{attribute addProperty BoxType "EL2262--0000"}
{attribute addProperty Id "OutputAT %Q*BYTE81"}
{attribute addProperty CRC "798999389"}
{attribute addProperty SizeInBites "8"}
{attribute addProperty SizeInBytes "1"}
TYPE Sample_2F9FC35D :
STRUCT
	{attribute addProperty Name "Output"}
	Output AT %Q* : BYTE;
END_STRUCT
END_TYPE

(* stored: Version 1.2.0.0, ProductVersion 3.1.4024.9
   DUT Sample_2F9FC35D: Id {000878ed-6930-43ab-ad1a-568c42e78b6e} *)
